// TIA Portal V19 export
FUNCTION "FC20_HmiLight" : Void   // FC20, LAD
{ S7_Optimized_Access := 'TRUE' }
// stored: AutoNumber false, IsIECCheckEnabled true, SetENOAutomatically false
   VAR_TEMP
      txStartUpWarning : Bool;
      txFaultError : Bool;
      txConditionOk : Bool;
      txReqOperator : Bool;
   END_VAR
   VAR CONSTANT
      cusiAutoMode : USInt := 1;   // Automatic mode
      cusiSemiAutoMode : USInt := 3;   // Semi-Automatic mode
      cusiMaintenanceMode : USInt := 2;   // Maintenance mode
   END_VAR
   VAR_TEMP   // added for the SCL form of the ladder/FBD networks
      _w1 : Bool;
      _w2 : Bool;
   END_VAR
BEGIN

REGION Network 1: Commande reset general
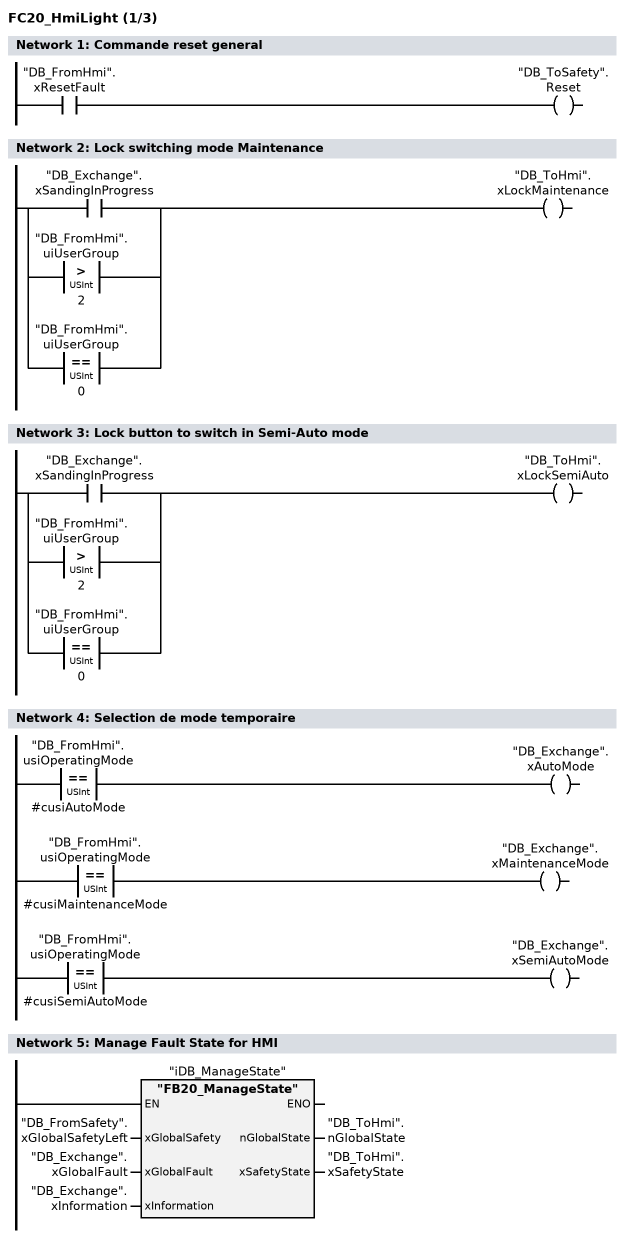
   RUNG wire#powerrail
      Contact( "DB_FromHmi".xResetFault )
      Coil( "DB_ToSafety".Reset )
   END_RUNG
   // the same network as SCL:
   "DB_ToSafety".Reset := "DB_FromHmi".xResetFault;
END_REGION

REGION Network 2: Lock switching mode Maintenance
   RUNG wire#powerrail
      Contact( "DB_Exchange".xSandingInProgress )
      wire#w1
      Coil( "DB_ToHmi".xLockMaintenance )
   END_RUNG
   RUNG wire#powerrail
      { S7_Templates := "SrcType := USInt" } GT_Contact(in1 := "DB_FromHmi".uiUserGroup, in2 := 2)
   END_RUNG wire#w1
   RUNG wire#powerrail
      { S7_Templates := "SrcType := USInt" } EQ_Contact(in1 := "DB_FromHmi".uiUserGroup, in2 := 0)
   END_RUNG wire#w1
   // the same network as SCL:
   "DB_ToHmi".xLockMaintenance := "DB_Exchange".xSandingInProgress OR ("DB_FromHmi".uiUserGroup > 2) OR ("DB_FromHmi".uiUserGroup = 0);
END_REGION

REGION Network 3: Lock button to switch in Semi-Auto mode
   RUNG wire#powerrail
      Contact( "DB_Exchange".xSandingInProgress )
      wire#w1
      Coil( "DB_ToHmi".xLockSemiAuto )
   END_RUNG
   RUNG wire#powerrail
      { S7_Templates := "SrcType := USInt" } GT_Contact(in1 := "DB_FromHmi".uiUserGroup, in2 := 2)
   END_RUNG wire#w1
   RUNG wire#powerrail
      { S7_Templates := "SrcType := USInt" } EQ_Contact(in1 := "DB_FromHmi".uiUserGroup, in2 := 0)
   END_RUNG wire#w1
   // the same network as SCL:
   "DB_ToHmi".xLockSemiAuto := "DB_Exchange".xSandingInProgress OR ("DB_FromHmi".uiUserGroup > 2) OR ("DB_FromHmi".uiUserGroup = 0);
END_REGION

REGION Network 4: Selection de mode temporaire
   RUNG wire#powerrail
      { S7_Templates := "SrcType := USInt" } EQ_Contact(in1 := "DB_FromHmi".usiOperatingMode, in2 := #cusiAutoMode)
      Coil( "DB_Exchange".xAutoMode )
   END_RUNG
   RUNG wire#powerrail
      { S7_Templates := "SrcType := USInt" } EQ_Contact(in1 := "DB_FromHmi".usiOperatingMode, in2 := #cusiMaintenanceMode)
      Coil( "DB_Exchange".xMaintenanceMode )
   END_RUNG
   RUNG wire#powerrail
      { S7_Templates := "SrcType := USInt" } EQ_Contact(in1 := "DB_FromHmi".usiOperatingMode, in2 := #cusiSemiAutoMode)
      Coil( "DB_Exchange".xSemiAutoMode )
   END_RUNG
   // the same network as SCL:
   "DB_Exchange".xAutoMode := "DB_FromHmi".usiOperatingMode = #cusiAutoMode;
   "DB_Exchange".xMaintenanceMode := "DB_FromHmi".usiOperatingMode = #cusiMaintenanceMode;
   "DB_Exchange".xSemiAutoMode := "DB_FromHmi".usiOperatingMode = #cusiSemiAutoMode;
END_REGION

REGION Network 5: Manage Fault State for HMI
   RUNG wire#powerrail
      "iDB_ManageState"(xGlobalSafety := "DB_FromSafety".xGlobalSafetyLeft, xGlobalFault := "DB_Exchange".xGlobalFault, xInformation := "DB_Exchange".xInformation, nGlobalState => "DB_ToHmi".nGlobalState, xSafetyState => "DB_ToHmi".xSafetyState)
   END_RUNG
   // the same network as SCL:
   "iDB_ManageState"(xGlobalSafety := "DB_FromSafety".xGlobalSafetyLeft,   // "FB20_ManageState"
                     xGlobalFault := "DB_Exchange".xGlobalFault,
                     xInformation := "DB_Exchange".xInformation,
                     nGlobalState => "DB_ToHmi".nGlobalState,
                     xSafetyState => "DB_ToHmi".xSafetyState);
END_REGION

REGION Network 6: Strat up warning
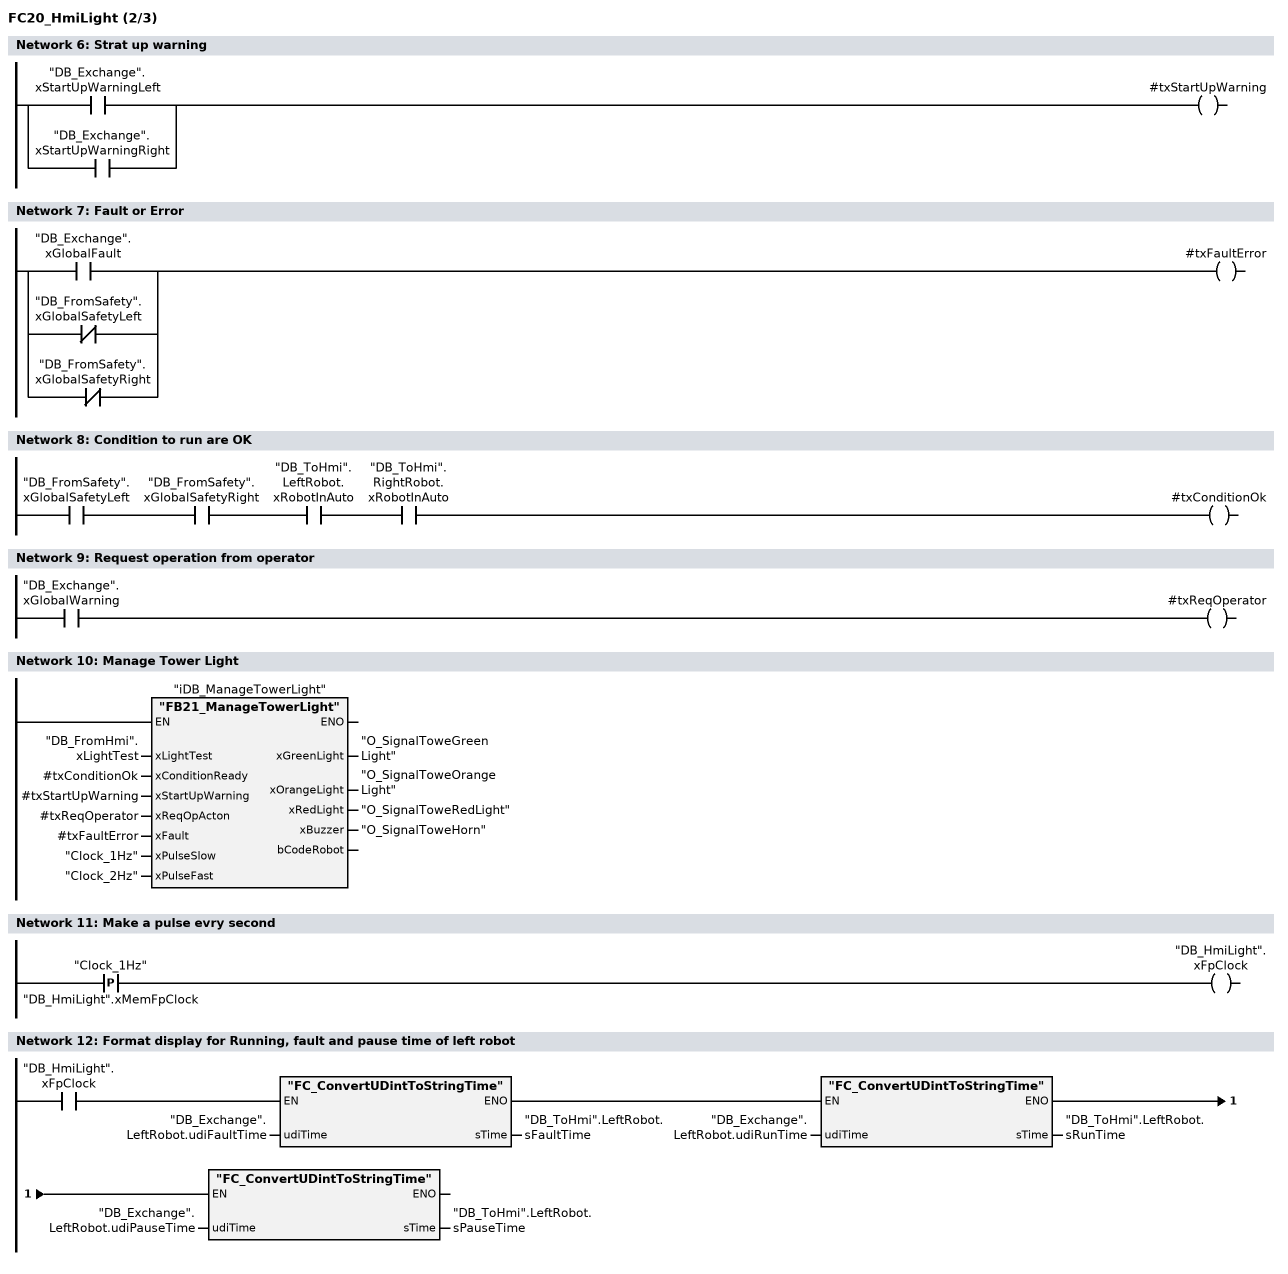
   RUNG wire#powerrail
      Contact( "DB_Exchange".xStartUpWarningLeft )
      wire#w1
      Coil( #txStartUpWarning )
   END_RUNG
   RUNG wire#powerrail
      Contact( "DB_Exchange".xStartUpWarningRight )
   END_RUNG wire#w1
   // the same network as SCL:
   #txStartUpWarning := "DB_Exchange".xStartUpWarningLeft OR "DB_Exchange".xStartUpWarningRight;
END_REGION

REGION Network 7: Fault or Error
   RUNG wire#powerrail
      Contact( "DB_Exchange".xGlobalFault )
      wire#w1
      Coil( #txFaultError )
   END_RUNG
   RUNG wire#powerrail
      I_Contact( "DB_FromSafety".xGlobalSafetyLeft )
   END_RUNG wire#w1
   RUNG wire#powerrail
      I_Contact( "DB_FromSafety".xGlobalSafetyRight )
   END_RUNG wire#w1
   // the same network as SCL:
   #txFaultError := "DB_Exchange".xGlobalFault OR NOT "DB_FromSafety".xGlobalSafetyLeft OR NOT "DB_FromSafety".xGlobalSafetyRight;
END_REGION

REGION Network 8: Condition to run are OK
   RUNG wire#powerrail
      Contact( "DB_FromSafety".xGlobalSafetyLeft )
      Contact( "DB_FromSafety".xGlobalSafetyRight )
      Contact( "DB_ToHmi".LeftRobot.xRobotInAuto )
      Contact( "DB_ToHmi".RightRobot.xRobotInAuto )
      Coil( #txConditionOk )
   END_RUNG
   // the same network as SCL:
   #txConditionOk := "DB_FromSafety".xGlobalSafetyLeft AND "DB_FromSafety".xGlobalSafetyRight AND "DB_ToHmi".LeftRobot.xRobotInAuto AND "DB_ToHmi".RightRobot.xRobotInAuto;
END_REGION

REGION Network 9: Request operation from operator
   RUNG wire#powerrail
      Contact( "DB_Exchange".xGlobalWarning )
      Coil( #txReqOperator )
   END_RUNG
   // the same network as SCL:
   #txReqOperator := "DB_Exchange".xGlobalWarning;
END_REGION

REGION Network 10: Manage Tower Light
   RUNG wire#powerrail
      "iDB_ManageTowerLight"(xLightTest := "DB_FromHmi".xLightTest, xConditionReady := #txConditionOk, xStartUpWarning := #txStartUpWarning, xReqOpActon := #txReqOperator, xFault := #txFaultError, xPulseSlow := "Clock_1Hz", xPulseFast := "Clock_2Hz", xGreenLight => "O_SignalToweGreenLight", xOrangeLight => "O_SignalToweOrangeLight", xRedLight => "O_SignalToweRedLight", xBuzzer => "O_SignalToweHorn", bCodeRobot =>)
   END_RUNG
   // the same network as SCL:
   "iDB_ManageTowerLight"(xLightTest := "DB_FromHmi".xLightTest,   // "FB21_ManageTowerLight"
                          xConditionReady := #txConditionOk,
                          xStartUpWarning := #txStartUpWarning,
                          xReqOpActon := #txReqOperator,
                          xFault := #txFaultError,
                          xPulseSlow := "Clock_1Hz",
                          xPulseFast := "Clock_2Hz",
                          xGreenLight => "O_SignalToweGreenLight",
                          xOrangeLight => "O_SignalToweOrangeLight",
                          xRedLight => "O_SignalToweRedLight",
                          xBuzzer => "O_SignalToweHorn");
END_REGION

REGION Network 11: Make a pulse evry second
   RUNG wire#powerrail
      P_Contact(operand := "Clock_1Hz", bit := "DB_HmiLight".xMemFpClock)
      Coil( "DB_HmiLight".xFpClock )
   END_RUNG
   // the same network as SCL:
   #_w1 := "Clock_1Hz" AND NOT "DB_HmiLight".xMemFpClock;   // rising edge of "Clock_1Hz"
   "DB_HmiLight".xMemFpClock := "Clock_1Hz";
   "DB_HmiLight".xFpClock := #_w1;
END_REGION

REGION Network 12: Format display for Running, fault and pause time of left robot
   RUNG wire#powerrail
      Contact( "DB_HmiLight".xFpClock )
      "FC_ConvertUDintToStringTime"(udiTime := "DB_Exchange".LeftRobot.udiFaultTime, sTime => "DB_ToHmi".LeftRobot.sFaultTime)
      "FC_ConvertUDintToStringTime"(udiTime := "DB_Exchange".LeftRobot.udiRunTime, sTime => "DB_ToHmi".LeftRobot.sRunTime)
      "FC_ConvertUDintToStringTime"(udiTime := "DB_Exchange".LeftRobot.udiPauseTime, sTime => "DB_ToHmi".LeftRobot.sPauseTime)
   END_RUNG
   // the same network as SCL:
   "FC_ConvertUDintToStringTime"(EN := "DB_HmiLight".xFpClock,
                           udiTime := "DB_Exchange".LeftRobot.udiFaultTime,
                           sTime => "DB_ToHmi".LeftRobot.sFaultTime,
                           ENO => #_w1);
   "FC_ConvertUDintToStringTime"(EN := #_w1,
                           udiTime := "DB_Exchange".LeftRobot.udiRunTime,
                           sTime => "DB_ToHmi".LeftRobot.sRunTime,
                           ENO => #_w2);
   IF #_w2 THEN
       "FC_ConvertUDintToStringTime"(udiTime := "DB_Exchange".LeftRobot.udiPauseTime,
                               sTime => "DB_ToHmi".LeftRobot.sPauseTime);
   END_IF;
END_REGION

REGION Network 13: Format display for Robot power on et robto drive on time of left robot
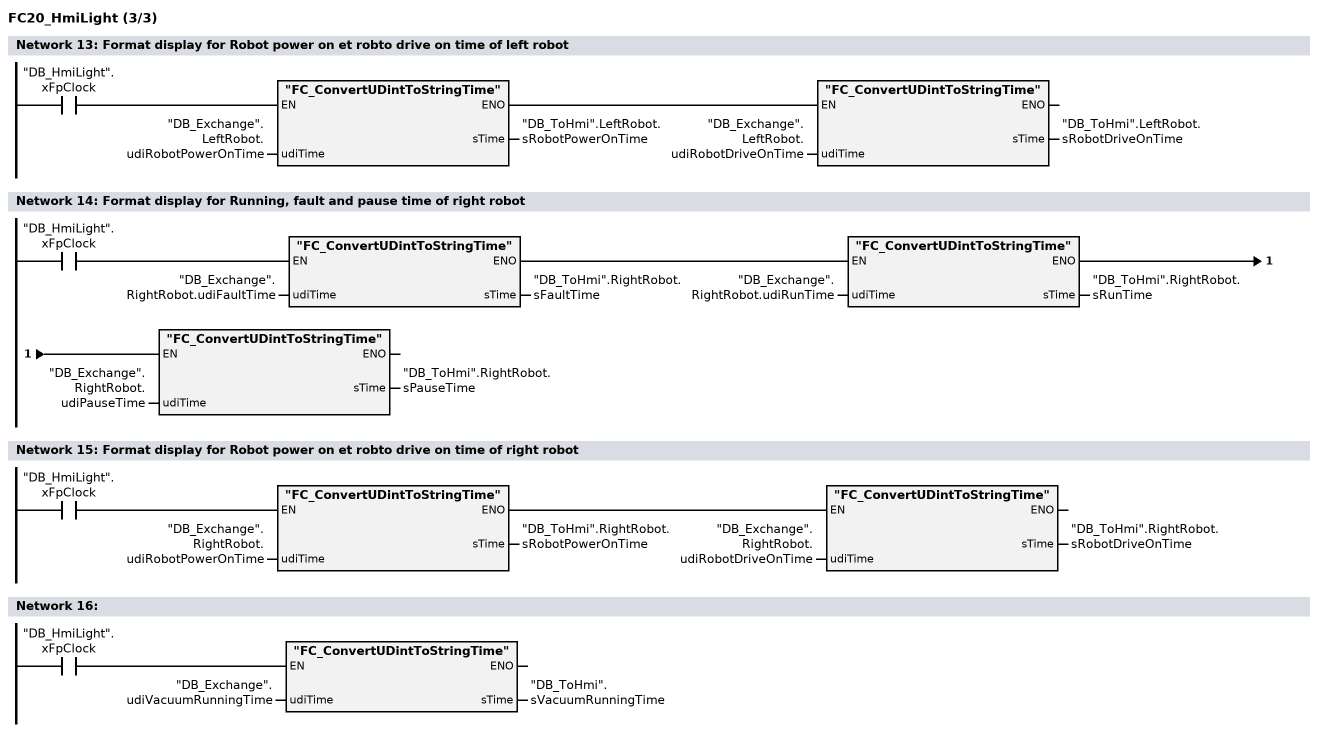
   RUNG wire#powerrail
      Contact( "DB_HmiLight".xFpClock )
      "FC_ConvertUDintToStringTime"(udiTime := "DB_Exchange".LeftRobot.udiRobotPowerOnTime, sTime => "DB_ToHmi".LeftRobot.sRobotPowerOnTime)
      "FC_ConvertUDintToStringTime"(udiTime := "DB_Exchange".LeftRobot.udiRobotDriveOnTime, sTime => "DB_ToHmi".LeftRobot.sRobotDriveOnTime)
   END_RUNG
   // the same network as SCL:
   "FC_ConvertUDintToStringTime"(EN := "DB_HmiLight".xFpClock,
                           udiTime := "DB_Exchange".LeftRobot.udiRobotPowerOnTime,
                           sTime => "DB_ToHmi".LeftRobot.sRobotPowerOnTime,
                           ENO => #_w1);
   IF #_w1 THEN
       "FC_ConvertUDintToStringTime"(udiTime := "DB_Exchange".LeftRobot.udiRobotDriveOnTime,
                               sTime => "DB_ToHmi".LeftRobot.sRobotDriveOnTime);
   END_IF;
END_REGION

REGION Network 14: Format display for Running, fault and pause time of right robot
   RUNG wire#powerrail
      Contact( "DB_HmiLight".xFpClock )
      "FC_ConvertUDintToStringTime"(udiTime := "DB_Exchange".RightRobot.udiFaultTime, sTime => "DB_ToHmi".RightRobot.sFaultTime)
      "FC_ConvertUDintToStringTime"(udiTime := "DB_Exchange".RightRobot.udiRunTime, sTime => "DB_ToHmi".RightRobot.sRunTime)
      "FC_ConvertUDintToStringTime"(udiTime := "DB_Exchange".RightRobot.udiPauseTime, sTime => "DB_ToHmi".RightRobot.sPauseTime)
   END_RUNG
   // the same network as SCL:
   "FC_ConvertUDintToStringTime"(EN := "DB_HmiLight".xFpClock,
                           udiTime := "DB_Exchange".RightRobot.udiFaultTime,
                           sTime => "DB_ToHmi".RightRobot.sFaultTime,
                           ENO => #_w1);
   "FC_ConvertUDintToStringTime"(EN := #_w1,
                           udiTime := "DB_Exchange".RightRobot.udiRunTime,
                           sTime => "DB_ToHmi".RightRobot.sRunTime,
                           ENO => #_w2);
   IF #_w2 THEN
       "FC_ConvertUDintToStringTime"(udiTime := "DB_Exchange".RightRobot.udiPauseTime,
                               sTime => "DB_ToHmi".RightRobot.sPauseTime);
   END_IF;
END_REGION

REGION Network 15: Format display for Robot power on et robto drive on time of right robot
   RUNG wire#powerrail
      Contact( "DB_HmiLight".xFpClock )
      "FC_ConvertUDintToStringTime"(udiTime := "DB_Exchange".RightRobot.udiRobotPowerOnTime, sTime => "DB_ToHmi".RightRobot.sRobotPowerOnTime)
      "FC_ConvertUDintToStringTime"(udiTime := "DB_Exchange".RightRobot.udiRobotDriveOnTime, sTime => "DB_ToHmi".RightRobot.sRobotDriveOnTime)
   END_RUNG
   // the same network as SCL:
   "FC_ConvertUDintToStringTime"(EN := "DB_HmiLight".xFpClock,
                           udiTime := "DB_Exchange".RightRobot.udiRobotPowerOnTime,
                           sTime => "DB_ToHmi".RightRobot.sRobotPowerOnTime,
                           ENO => #_w1);
   IF #_w1 THEN
       "FC_ConvertUDintToStringTime"(udiTime := "DB_Exchange".RightRobot.udiRobotDriveOnTime,
                               sTime => "DB_ToHmi".RightRobot.sRobotDriveOnTime);
   END_IF;
END_REGION

REGION Network 16
   RUNG wire#powerrail
      Contact( "DB_HmiLight".xFpClock )
      "FC_ConvertUDintToStringTime"(udiTime := "DB_Exchange".udiVacuumRunningTime, sTime => "DB_ToHmi".sVacuumRunningTime)
   END_RUNG
   // the same network as SCL:
   IF "DB_HmiLight".xFpClock THEN
       "FC_ConvertUDintToStringTime"(udiTime := "DB_Exchange".udiVacuumRunningTime,
                               sTime => "DB_ToHmi".sVacuumRunningTime);
   END_IF;
END_REGION

REGION Network 17 (SCL): Copy status to HMI
   "DB_ToHmi".xAccessDoor := "DB_FromSafety".DoorAcces.State;
   "DB_ToHmi".xCaptiveKey := "DB_FromSafety".CaptiveKeyInLock.State;
   "DB_ToHmi".xLightBeam := "DB_FromSafety".PedestrialDoorAcces.State;
   "DB_ToHmi".xCbsGate := "DB_FromSafety".GateAccesCBS.State;
END_REGION
END_FUNCTION
